// Block: TRK_Info

DATA_BLOCK TRK_Info
VERSION : 0.1
   NON_RETAIN
   VAR
      HMI_Info : BTrk_item;
   END_VAR

BEGIN
   // No initialization required
END_DATA_BLOCK
